// TIA Portal V19 export
ORGANIZATION_BLOCK "IO"   // OB123, FBD, ProgramCycle
TITLE = "Main Program Sweep (Cycle)"
{ S7_Optimized_Access := 'TRUE' }
// stored: SetENOAutomatically false
   VAR_INPUT
      Initial_Call : Bool;   // Initial call of this OB
      Remanence : Bool;   // =True, if remanent data are available
   END_VAR
   VAR_TEMP
      "101CV1_Temp" : Real;
      "101CV2_Temp" : Real;
   END_VAR
   VAR_TEMP   // added for the SCL form of the ladder/FBD networks
      _w1 : Bool;
   END_VAR
BEGIN

REGION Network 1
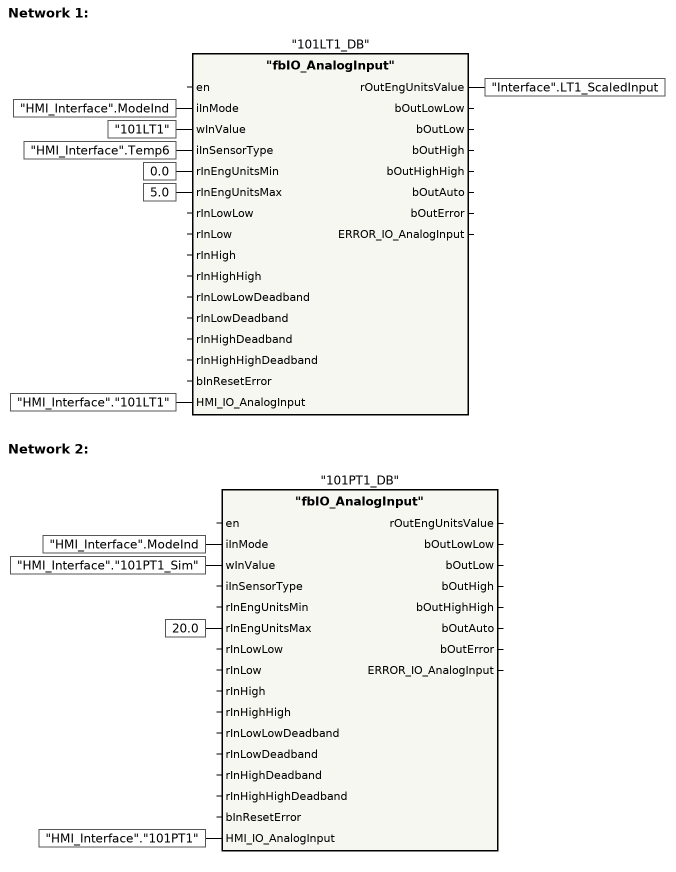
   "101LT1_DB"(iInMode := "HMI_Interface".ModeInd,   // "fbIO_AnalogInput"
               wInValue := "101LT1",
               iInSensorType := "HMI_Interface".Temp6,
               rInEngUnitsMin := 0.0,
               rInEngUnitsMax := 5.0,
               HMI_IO_AnalogInput := "HMI_Interface"."101LT1",
               rOutEngUnitsValue => "Interface".LT1_ScaledInput);
END_REGION

REGION Network 2
   "101PT1_DB"(iInMode := "HMI_Interface".ModeInd,   // "fbIO_AnalogInput"
               wInValue := "HMI_Interface"."101PT1_Sim",
               rInEngUnitsMax := 20.0,
               HMI_IO_AnalogInput := "HMI_Interface"."101PT1");
END_REGION

REGION Network 3: "101CV1
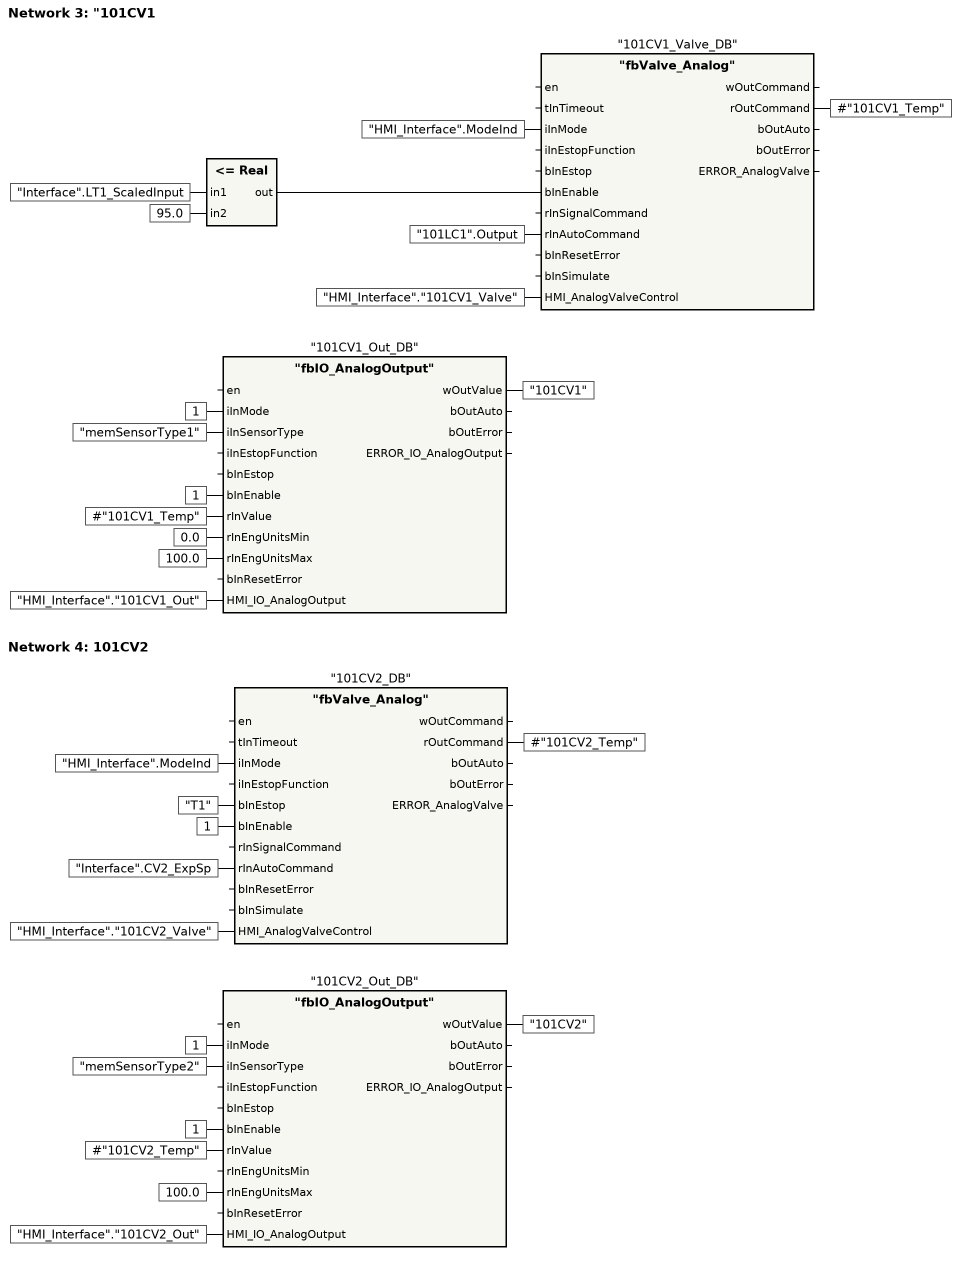
   "101CV1_Valve_DB"(iInMode := "HMI_Interface".ModeInd,   // "fbValve_Analog"
                     bInEnable := "Interface".LT1_ScaledInput <= 95.0,
                     rInAutoCommand := "101LC1".Output,
                     HMI_AnalogValveControl := "HMI_Interface"."101CV1_Valve",
                     rOutCommand => #"101CV1_Temp");
   "101CV1_Out_DB"(iInMode := 1,   // "fbIO_AnalogOutput"
                   iInSensorType := "memSensorType1",
                   bInEnable := 1,
                   rInValue := #"101CV1_Temp",
                   rInEngUnitsMin := 0.0,
                   rInEngUnitsMax := 100.0,
                   HMI_IO_AnalogOutput := "HMI_Interface"."101CV1_Out",
                   wOutValue => "101CV1");
END_REGION

REGION Network 4: 101CV2
   "101CV2_DB"(iInMode := "HMI_Interface".ModeInd,   // "fbValve_Analog"
               bInEstop := "T1",
               bInEnable := 1,
               rInAutoCommand := "Interface".CV2_ExpSp,
               HMI_AnalogValveControl := "HMI_Interface"."101CV2_Valve",
               rOutCommand => #"101CV2_Temp");
   "101CV2_Out_DB"(iInMode := 1,   // "fbIO_AnalogOutput"
                   iInSensorType := "memSensorType2",
                   bInEnable := 1,
                   rInValue := #"101CV2_Temp",
                   rInEngUnitsMax := 100.0,
                   HMI_IO_AnalogOutput := "HMI_Interface"."101CV2_Out",
                   wOutValue => "101CV2");
END_REGION

REGION Network 5: 101DV1
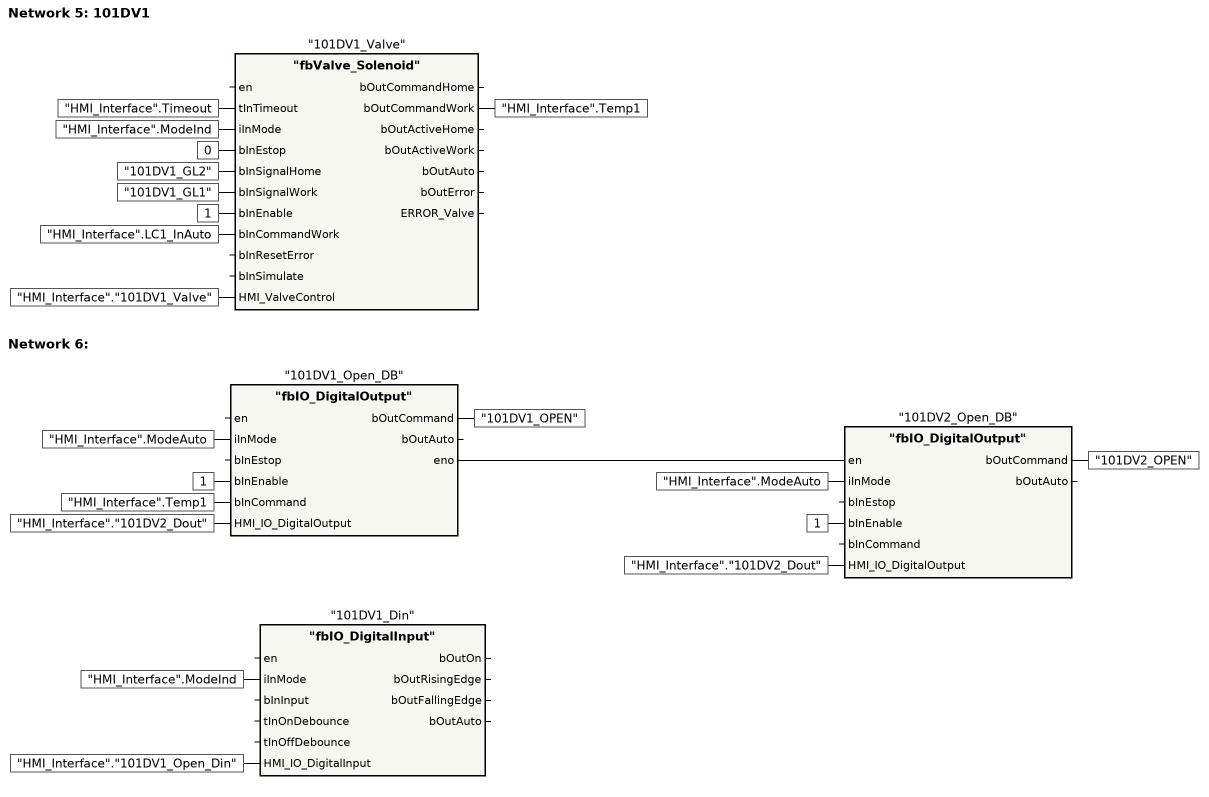
   "101DV1_Valve"(tInTimeout := "HMI_Interface".Timeout,   // "fbValve_Solenoid"
                  iInMode := "HMI_Interface".ModeInd,
                  bInEstop := 0,
                  bInSignalHome := "101DV1_GL2",
                  bInSignalWork := "101DV1_GL1",
                  bInEnable := 1,
                  bInCommandWork := "HMI_Interface".LC1_InAuto,
                  HMI_ValveControl := "HMI_Interface"."101DV1_Valve",
                  bOutCommandWork => "HMI_Interface".Temp1);
END_REGION

REGION Network 6
   "101DV1_Open_DB"(iInMode := "HMI_Interface".ModeAuto,   // "fbIO_DigitalOutput"
                    bInEnable := 1,
                    bInCommand := "HMI_Interface".Temp1,
                    HMI_IO_DigitalOutput := "HMI_Interface"."101DV2_Dout",
                    bOutCommand => "101DV1_OPEN",
                    ENO => #_w1);
   IF #_w1 THEN
       "101DV2_Open_DB"(iInMode := "HMI_Interface".ModeAuto,   // "fbIO_DigitalOutput"
                        bInEnable := 1,
                        HMI_IO_DigitalOutput := "HMI_Interface"."101DV2_Dout",
                        bOutCommand => "101DV2_OPEN");
   END_IF;
   "101DV1_Din"(iInMode := "HMI_Interface".ModeInd, HMI_IO_DigitalInput := "HMI_Interface"."101DV1_Open_Din");   // "fbIO_DigitalInput"
END_REGION
END_ORGANIZATION_BLOCK
